# EPICS autosave request: iocBoot/gmca_23i_ioc2/dbSave/JET_Ps_.req
%
% BURT Request File
%
% $(P)JET:Ps:  CryoJet positioner
%

file assy.req ASSY=$(P)JET:Ps
file mtr1.req MTR1=$(P)JET:mp
file drv1.req DRV1=$(P)JET:P
